FUNCTION_BLOCK CountCurrentPosition1
VAR_INPUT
END_VAR
VAR_OUTPUT
END_VAR
VAR
END_VAR

IF IO.Initialized THEN
	
	// COUNT ROTATION:
	IF IO.StepRotatonSwitch = 1 AND Automatic.RCurrentlyMoving THEN
		// away from the sensor:
		IF IO.MotorRotationDirection = 0 THEN
			IF (NOT IO.Switch) THEN		// in automatic mode
				IF IO.PreviousManualMode THEN	
					Automatic.RotationPositionCurrent := Automatic.RotationPositionCurrent + 1;
				ELSE	// to restore the state
					Automatic.RotationPositionCurrent := Automatic.RotationPositionCurrent + 1;
					Automatic.RotationPositionAuto := Automatic.RotationPositionAuto + 1;
				END_IF
			ELSE		// in manual mode
				Automatic.RotationPositionCurrent := Automatic.RotationPositionCurrent + 1;
			END_IF
		// towards the sensor:
		ELSE
			IF (NOT IO.Switch) THEN		// in automatic mode
				IF IO.PreviousManualMode THEN	
					Automatic.RotationPositionCurrent := Automatic.RotationPositionCurrent - 1;
				ELSE	// to restore the state
					Automatic.RotationPositionCurrent := Automatic.RotationPositionCurrent - 1;
					Automatic.RotationPositionAuto := Automatic.RotationPositionAuto - 1;
				END_IF
			ELSE		// in manual mode
				Automatic.RotationPositionCurrent := Automatic.RotationPositionCurrent - 1;
			END_IF
		END_IF
	END_IF
	
	// COUNT Extension: (-------edino še NESPREMENJENO--------)
	IF IO.StepExtensionSwitch = 1 THEN
		IF IO.MotorExtensionDirection = 0 THEN
			IF (NOT IO.Switch) AND Automatic.ECurrentlyMoving THEN
				IF IO.PreviousManualMode THEN
					Automatic.ExtensionPositionCurrent := Automatic.ExtensionPositionCurrent + 1;
				ELSE
					Automatic.ExtensionPositionAuto := Automatic.ExtensionPositionAuto + 1;
					Automatic.ExtensionPositionCurrent := Automatic.ExtensionPositionCurrent + 1;
				END_IF
			ELSIF Automatic.ECurrentlyMoving THEN
				Automatic.ExtensionPositionCurrent := Automatic.ExtensionPositionCurrent + 1;
			END_IF
		ELSE
			IF (NOT IO.Switch) AND Automatic.ECurrentlyMoving THEN
				IF IO.PreviousManualMode THEN
					Automatic.ExtensionPositionCurrent := Automatic.ExtensionPositionCurrent - 1;
				ELSE
					Automatic.ExtensionPositionAuto := Automatic.ExtensionPositionAuto - 1;
					Automatic.ExtensionPositionCurrent := Automatic.ExtensionPositionCurrent - 1;
				END_IF
			ELSIF Automatic.ECurrentlyMoving THEN
				Automatic.ExtensionPositionCurrent := Automatic.ExtensionPositionCurrent - 1;
			END_IF
		END_IF
	END_IF
	
	// COUNT Lifting:
	IF IO.StepLiftingSwitch = 1 AND Automatic.LCurrentlyMoving THEN
		// away from the sensor:
		IF IO.MotorLiftingDirection = 0 THEN
			IF (NOT IO.Switch) THEN		// in automatic mode
				IF IO.PreviousManualMode THEN
					Automatic.LiftingPositionCurrent := Automatic.LiftingPositionCurrent + 1;
				ELSE	// to restore the state
					Automatic.LiftingPositionCurrent := Automatic.LiftingPositionCurrent + 1;
					Automatic.LiftingPositionAuto := Automatic.LiftingPositionAuto + 1;
				END_IF
			ELSE		// in manual mode
				Automatic.LiftingPositionCurrent := Automatic.LiftingPositionCurrent + 1;
			END_IF
		// towards the sensor:
		ELSE
			IF (NOT IO.Switch) THEN		// in automatic mode
				IF IO.PreviousManualMode THEN
					Automatic.LiftingPositionCurrent := Automatic.LiftingPositionCurrent - 1;
				ELSE	// to restore the state
					Automatic.LiftingPositionAuto := Automatic.LiftingPositionAuto - 1;
					Automatic.LiftingPositionCurrent := Automatic.LiftingPositionCurrent - 1;
				END_IF
			ELSE		// in manual mode
				Automatic.LiftingPositionCurrent := Automatic.LiftingPositionCurrent - 1;
			END_IF
		END_IF
	END_IF
	
	// COUNT Grip:
	IF IO.StepGripSwitch = 1 AND Automatic.GCurrentlyMoving THEN
		IF IO.MotorGripDirection = 0 THEN
			IF (NOT IO.Switch) THEN		// in automatic mode
				IF IO.PreviousManualMode THEN
					Automatic.GripPositionCurrent := Automatic.GripPositionCurrent + 1;
				ELSE
					Automatic.GripPositionAuto := Automatic.GripPositionAuto + 1;
					Automatic.GripPositionCurrent := Automatic.GripPositionCurrent + 1;
				END_IF
			ELSE		// in manual mode
				Automatic.GripPositionCurrent := Automatic.GripPositionCurrent + 1;
			END_IF
		ELSE
			IF (NOT IO.Switch) THEN		// in automatic mode
				IF IO.PreviousManualMode THEN
					Automatic.GripPositionCurrent := Automatic.GripPositionCurrent - 1;
				ELSE
					Automatic.GripPositionAuto := Automatic.GripPositionAuto - 1;
					Automatic.GripPositionCurrent := Automatic.GripPositionCurrent - 1;
				END_IF
			ELSE		// in manual mode
				Automatic.GripPositionCurrent := Automatic.GripPositionCurrent - 1;
			END_IF
		END_IF
	END_IF
	
END_IF

END_FUNCTION_BLOCK

(* stored: Version 1.1.0.1, ProductVersion 3.1.4024.13
   POU CountCurrentPosition1: Id {9470ef1e-6d57-4400-87bd-bf87707256a6}, SpecialFunc None *)
